// TIA Portal V20 export
// export: Created 2025-12-01T14:57:08.1676699Z, ExportSetting None, DisplayName Totally Integrated Automation Portal, DisplayVersion V20 Update 3, DisplayName TIA Portal Openness, DisplayVersion V20 Update 3, DisplayName TIA Portal Version Control Interface, DisplayVersion V20 Update 3, DisplayName STEP 7 Professional, DisplayVersion V20 Update 3, DisplayName STEP 7 Safety, DisplayVersion V20 Update 2, DisplayName WinCC Basic/Comfort/Advanced, DisplayVersion V20 Update 3, DisplayName WinCC Professional, DisplayVersion V20 Update 3, DisplayName WinCC Unified, DisplayVersion V20 Update 3
FUNCTION "FC860_Informe_DatosUT" : Void   // FC860, STL
{ S7_Optimized_Access := 'FALSE' }
// stored: AutoNumber false
   VAR_INPUT
      Mesa : UInt;
   END_VAR
   VAR_OUTPUT
      Informe_DatosUT : "UDT_Informe_DatosUT";
   END_VAR
   VAR_TEMP
      NumeroUT : Int;
      Relleno : Byte;
      ValorReturn : Int;
   END_VAR
BEGIN

NETWORK
TITLE = Inicializar
//////////////////////////////////////////////////////////////////////
/// Inicializar Variables

      L     0;
      T     #Relleno;

      CALL  FILL
      ( BVAL    := #Relleno,
        RET_VAL := #ValorReturn,
        BLK     := #Informe_DatosUT
      );



NETWORK
TITLE = Buscar Primera UT de la Mesa
//////////////////////////////////////////////////////////////////////
/// Buscar Primera UT de la Mesa
      L     "DB810_ColasMesas".Colas[#Mesa].UT_PrimeraMesa;
      T     #NumeroUT;

      L     #NumeroUT;
      L     0;
      <>I;
      JC    CrearInforme;

      BE;  // - Finalizar bloque



NETWORK
TITLE = Crear Informe
CrearInforme:NOP   0;

//////////////////////////////////////////////////////////////////////
/// Crear Informe de la UT

      L     "DB812_UTs_Control".UT[#NumeroUT].MesaDestino;
      T     #Informe_DatosUT.MesaDestino;

      L     "DB812_UTs_Control".UT[#NumeroUT].TipoCarga;
      T     #Informe_DatosUT.TipoCarga;

      SET;
      A     "DB812_UTs_Control".UT[#NumeroUT].AtributosDelaCarga.Vacia;
      =     #Informe_DatosUT.AtributosCarga.Vacia;
      SET;
      A     "DB812_UTs_Control".UT[#NumeroUT].AtributosDelaCarga.Pila;
      =     #Informe_DatosUT.AtributosCarga.Pila;
      SET;
      A     "DB812_UTs_Control".UT[#NumeroUT].AtributosDelaCarga.Remontada;
      =     #Informe_DatosUT.AtributosCarga.Remontada;


      L     "DB815_UTs_Datos".UT[#NumeroUT].CodigoEnfardado;
      T     #Informe_DatosUT.Enfradado;
      L     "DB815_UTs_Datos".UT[#NumeroUT].CodigoFlejado;
      T     #Informe_DatosUT.Flejado;
      L     "DB815_UTs_Datos".UT[#NumeroUT].CodigoEtiquetado;
      T     #Informe_DatosUT.Etiquetado;

      L     "DB815_UTs_Datos".UT[#NumeroUT].CotaAltura;
      T     #Informe_DatosUT.CotaAltura;
      L     "DB815_UTs_Datos".UT[#NumeroUT].CotaAnchura;
      T     #Informe_DatosUT.CotaAnchura;
      L     "DB815_UTs_Datos".UT[#NumeroUT].CotaProfundidad;
      T     #Informe_DatosUT.CotaLargura;

      L     "DB815_UTs_Datos".UT[#NumeroUT].Peso;
      T     #Informe_DatosUT.Peso;

      SET;
      A     "DB812_UTs_Control".UT[#NumeroUT].AtributosDeLaUT.LadoDeLaEtiqueta;
      =     #Informe_DatosUT.PosEtiqueta.Derecha;

      SET;
      AN    "DB812_UTs_Control".UT[#NumeroUT].AtributosDeLaUT.LadoDeLaEtiqueta;
      =     #Informe_DatosUT.PosEtiqueta.Izquierda;

// nieves añadido volcado de la información de las etiquetas

      CALL  MOVE
      ( IN  := "DB814_UTs_Etiqueta".UT[#NumeroUT].Etiqueta,
        OUT := #Informe_DatosUT.etiqueta
      );


      L     "DB814_UTs_Etiqueta".UT[#NumeroUT].EtiquetaRouter;
      T     #Informe_DatosUT.EtiquetaRouter;

// fin añadido nieves
      BE;  // - Finalizar bloque


END_FUNCTION
